FUNCTION_BLOCK FB_Listener EXTENDS FB_ListenerBase2
VAR_INPUT
	sSourceFilter			: STRING;	// filter events by this source
END_VAR

VAR_OUTPUT
	aStSavedEvents			: ARRAY [1..GVL_SafetyEvents.MAX_EVENTS] OF ST_Event;	// output array
END_VAR

VAR
	nCntMessagesSent		: UINT;		// messages sent counter
	nCntMessagesNow			: UINT;		// messages sent at once counter
	nCntMessagesSaved		: UINT;		// messages saved in output array counter
	
	nCntRequestReturn		: UINT;		// internal counter, used to delay output queue, and get event text before
	
	nIdx					: UINT;		// index, used in for loops
	
	bReqText				: ARRAY [1..GVL_SafetyEvents.MAX_CURR] OF BOOL;	// request event text flag
	
	aStCachedEvents			: ARRAY [1..GVL_SafetyEvents.MAX_CURR] OF ST_Event;	// cached event structure
	
	SystemTime				: T_FILETIME;						// system time structure
	fbGetSystemTime			: GETSYSTEMTIME;					// get system time fb
	fbRequestEventText		: ARRAY [1..GVL_SafetyEvents.MAX_CURR] OF FB_RequestEventText;	// request event text fb
END_VAR

METHOD ClearOutput : HRESULT
VAR_INPUT
END_VAR
MEMSET(ADR(aStSavedEvents), 16#00, SIZEOF(aStSavedEvents));
END_METHOD

METHOD Execute : HRESULT
// Retrieve events
Execute := SUPER^.Execute();

// Reset retrieved text counter
nCntRequestReturn := 0;

// Retrieve the text of queued messages
FOR nIdx := 1 TO nCntMessagesNow DO
	// If requested, and error
	IF 	bReqText[nIdx] AND fbRequestEventText[nIdx].bError THEN
		// Reset request flag
		bReqText[nIdx] := FALSE;
		// Show error message
		aStCachedEvents[nIdx].EventText := 'Error retrieve event text';
		nCntRequestReturn := nCntRequestReturn + 1;
	// If requested and retrieved
	ELSIF bReqText[nIdx] AND NOT fbRequestEventText[nIdx].bBusy THEN
		// Get retrieved text
		fbRequestEventText[nIdx].GetString(aStCachedEvents[nIdx].EventText, SIZEOF(aStCachedEvents[nIdx].EventText));
		// Reset request flag
		bReqText[nIdx] := FALSE;
		// Increase retrieved text counter
		nCntRequestReturn := nCntRequestReturn + 1;
	END_IF
END_FOR

// If catched events are present, and all requests are retrevied ...
IF nCntMessagesSent > nCntMessagesSaved AND nCntRequestReturn = nCntMessagesNow THEN
	// Reset catched events number
	nCntMessagesSaved := nCntMessagesSent;
	// Move output array
	MEMMOVE(ADR(aStSavedEvents[nCntMessagesNow + 1]), ADR(aStSavedEvents[1]), SIZEOF(aStSavedEvents[1]) * (GVL_SafetyEvents.MAX_CURR - nCntMessagesNow));
	// Move catched events to output array
	FOR nIdx := 1 TO nCntMessagesNow DO
		aStSavedEvents[nIdx] := aStCachedEvents[nIdx];
	END_FOR
	// Reset current catched events counter
	nCntMessagesNow := 0;
END_IF
END_METHOD

METHOD OnMessageSent : HRESULT

VAR_INPUT
	fbEvent : REFERENCE TO FB_TcEvent;
END_VAR
// If source is different that desired module, skip this event
IF fbEvent.ipSourceInfo.sName = sSourceFilter THEN
	// If possible, count handled events
	IF (nCntMessagesSent + 1) < 65535 THEN
		nCntMessagesSent	:= nCntMessagesSent + 1;
	// If counter overflow, reset counters and continue work ...
	ELSE
		nCntMessagesSent	:= 1;
		nCntMessagesSaved	:= 0;
	END_IF
	
	// If messages at once are less than max...
	IF nCntMessagesNow + 1 <= GVL_SafetyEvents.MAX_CURR THEN
		// Increase messages at once counter (if no delay between events, this method will be called more than once, so we use iterator to handle more events at once)
		nCntMessagesNow	:= nCntMessagesNow + 1;
		
		// Request event text
		fbRequestEventText[nCntMessagesNow].Request(
			eventClass	:= fbEvent.EventClass,
			nEventId	:= fbEvent.nEventId,
			nLangId		:= 1033,
			ipArgs		:= fbEvent.ipArguments
		);
		
		// Set request flag
		bReqText[nCntMessagesNow] := TRUE;
		
		// Save event data
		aStCachedEvents[nCntMessagesNow].EventID	:= fbEvent.nEventId;
		aStCachedEvents[nCntMessagesNow].Severity	:= TO_BYTE(fbEvent.eSeverity);
		
		// Get current system time
		fbGetSystemTime(
			timeLoDW => SystemTime.dwLowDateTime,
			timeHiDW => SystemTime.dwHighDateTime );
		
		// Save current system time, as event raised time
		aStCachedEvents[nCntMessagesNow].TimeRaised	:= FILETIME_TO_DT(SystemTime); // Convert time to DateTime format
	
		// Set output
		OnMessageSent	:= S_OK; // in order to receive more callbacks (Set <> S_OK in order to cancel the callbacks for this program cycle.)
	ELSE
		OnMessageSent	:= E_FAIL;
	END_IF
END_IF
END_METHOD

END_FUNCTION_BLOCK

(* stored: Version 1.1.0.1, ProductVersion 3.1.4024.4
   POU FB_Listener: Id {50ed088d-9a7d-4c16-86a9-e90b487e4982}, SpecialFunc None
   Method ClearOutput: Id {c8aa6c3c-f6bb-40db-bb62-da21a46514a8}
   Method Execute: Id {3c7f655d-2c73-41dc-b085-26c5a3b1cef1}
   Method OnMessageSent: Id {b4dac56d-cfe9-4434-ae5b-afa117054bdb} *)
